// TIA Portal V15.1 export
// export: Created 2022-03-15T12:28:27.7472711Z, ExportSetting WithDefaults, WithReadOnly, DisplayName Totally Integrated Automation Portal, DisplayVersion V15.1 Update 3, DisplayName TIA Portal Openness, DisplayVersion V15.1, DisplayName TIA Portal Teamcenter Gateway, DisplayVersion V15.1, DisplayName SINAMICS Startdrive Advanced, DisplayVersion V15.1, DisplayName G130, G150, S120, S150, SINAMICS MV, S210, DisplayVersion V15.1, DisplayName G110M, G120, G120C, G120D, G120P, DisplayVersion V15.1, DisplayName STEP 7 Professional, DisplayVersion V15.1 Update 3, DisplayName STEP 7 Safety, DisplayVersion V15.1, DisplayName WinCC Advanced, DisplayVersion V15.1 Update 3
FUNCTION_BLOCK "FB_Baustein_3"   // FB1, SCL
{ S7_Optimized_Access := 'TRUE' }
VERSION : 0.1
// stored: AutoNumber true, CodeModifiedDate 2022-03-08T11:13:52.8896608Z, CompileDate 2022-03-08T11:13:54.0933934Z, CreationDate 2022-03-08T11:12:33.2792339Z, DownloadWithoutReinit false, HandleErrorsWithinBlock false, InterfaceModifiedDate 2022-03-08T11:12:52.1304591Z, IsConsistent true, IsIECCheckEnabled false, IsKnowHowProtected false, ISMultiInstanceCapable true, IsRetainMemResEnabled false, IsWriteProtected false, LibraryConformanceStatus Das Objekt ist bibliothekskonform., MemoryReserve 100, ModifiedDate 2022-03-08T11:13:53.4529134Z, ParameterModified 2022-03-08T11:12:52.1304591Z, PLCSimAdvancedSupport false, SetENOAutomatically False, StructureModified 2022-03-08T11:12:52.1304591Z, UDAEnableTagReadback false
   VAR_INPUT
      Input_1 : Bool;
      Input_2 : Bool;
      Input_3 : Bool;
   END_VAR
   VAR_OUTPUT
      Output_1 : Bool;
      Output_2 : Bool;
      Output_3 : Bool;
   END_VAR
BEGIN
END_FUNCTION_BLOCK
